FUNCTION_BLOCK FB_Cell
VAR_INPUT
END_VAR
VAR_OUTPUT
END_VAR
VAR
	eAutoMan					: E_AutoMan := E_AutoMan.AUTO;
	State						: E_CellState;
	
	// IO
	bStartBtn					AT %I* : BOOL;
	bStopBtn					AT %I* : BOOL;
	bPartPresentAtInfeed		AT %I* : BOOL;
	bPartPresentAtOutfeed		AT %I* : BOOL;
	
	{attribute 'TcAnalytics'}
	fFillRate					AT %Q* : LREAL := 2.5;
	
	// devices
	fbInfeedActuator			: FB_Actuator;
	fbOutfeedActuator			: FB_Actuator;
	fbInfeedConveyor			: FB_Axis;
	fbIndexConveyor				: FB_Axis;
	fbOutfeedConveyor			: FB_Axis;
	
	InfeedConveyor				: IAxis := fbInfeedConveyor;
	IndexConveyor				: IAxis := fbIndexConveyor;
	InfeedActuator				: IActuator := fbInfeedActuator;
	OutfeedActuator				: IActuator := fbOutfeedActuator;
	OutfeedConveyor				: IAxis := fbOutfeedConveyor;
	
	// stations
	fbBarcoder					: FB_BarcodeScanner;
	fbFiller					: FB_Filler;
	fbCapper					: FB_Capper;
	fbCheckWeigher				: FB_CheckWeigher;
	Stations					: ARRAY[0..3] OF IStation := [fbBarcoder, fbFiller, fbCapper, fbCheckWeigher];
	iStationCount				: DINT := 4;
	i							: DINT;
	
	bAllStationsReady			: BOOL;
	bCellPartPresent			: BOOL;
	bStationFaulted				: BOOL;
	tmrStationWait				: TON;
	bInFeeding					: BOOL;
	bIndexing					: BOOL;
	bOutfeeding					: BOOL;
	
	PartStatus					: ARRAY[0..3] OF ST_PartStatus;
	NewPart						: ST_PartStatus;
	
	{attribute 'TcAnalytics'}
	OutfeedPart					: ST_PartStatus;
	
	fIndexPosition				: LREAL;
	INDEX_DIST					: LREAL := 300.0;
	INDEX_VEL					: LREAL := 100.0;
	INFEED_VEL					: LREAL := 100.0;
	
	bStartReq					: BOOL;
	bStopReq					: BOOL;
	bInit 						: BOOL := TRUE;
	
	bFillRateTest				: BOOL;
	tmrFillRate					: TON;
END_VAR

METHOD PUBLIC CheckPart : BOOL
VAR_INPUT
	Status			: ST_PartStatus;
END_VAR
CheckPart := Status.bBarcodeStatus AND Status.bFillerStatus AND Status.bCapperStatus AND Status.bWeightStatus;
END_METHOD

METHOD PUBLIC Execute : PVOID
StationMgr();

IF eAutoMan = E_AutoMan.AUTO THEN
	
	CASE State OF
		
		E_CellState.STOPPED:
			
			IF bStartReq THEN
				State := E_CellState.IDLE_WAIT;
				bStartReq := FALSE;
			END_IF
			
		E_CellState.IDLE_WAIT:
		
			IF bPartPresentAtInfeed AND Stations[0] <> 0 
			AND (Stations[0].Ready AND NOT Stations[0].PartPresent) THEN
				State := E_CellState.FEED;
			END_IF
			
			IF bAllStationsReady AND bCellPartPresent THEN
				tmrStationWait(IN:=TRUE, PT:=T#500MS);
				IF tmrStationWait.Q THEN
					tmrStationWait(IN:=FALSE);
					State := E_CellState.INDEX;
				END_IF
			END_IF
			
			IF bStopReq THEN
				State := E_CellState.STOPPED;
				bStopReq := FALSE;
			END_IF
			
		E_CellState.FEED:
		
			IF NOT bInFeeding THEN
				MEMCPY(ADR(PartStatus[0]), ADR(NewPart), SIZEOF(ST_PartStatus));
				bInFeeding := TRUE;
			END_IF
			
			IF InfeedActuator.Cycle() THEN
				State := E_CellState.IDLE_WAIT;
				bInFeeding := FALSE;
			END_IF
			
		E_CellState.INDEX:
			
			IF NOT bIndexing THEN
				fIndexPosition := IndexConveyor.ActPosition + INDEX_DIST;
				bIndexing := TRUE;
			END_IF
			
			IF (IndexConveyor.MoveAbsolute(fIndexPosition, INDEX_VEL)) AND bIndexing THEN
				bIndexing := FALSE;
				OutfeedPart := PartStatus[3];
				MEMCPY(ADR(PartStatus[1]), ADR(PartStatus[0]), SIZEOF(ST_PartStatus)*3);
				MEMSET(ADR(PartStatus[0]), 0, SIZEOF(ST_PartStatus));
				State := E_CellState.IDLE_WAIT;
			END_IF
			
	END_CASE
	
	IF State <> E_CellState.STOPPED THEN
		
		InfeedConveyor.JogFwd(INFEED_VEL);
		OutfeedConveyor.JogFwd(INFEED_VEL);
		
		IF bPartPresentAtOutfeed THEN
			// bad part
			IF NOT CheckPart(OutfeedPart) THEN
				bOutFeeding := TRUE;
			END_IF
		END_IF
		IF bOutfeeding THEN
			IF OutfeedActuator.Cycle() THEN
				bOutfeeding := FALSE;
			END_IF
		END_IF
		
		IF bFillRateTest THEN
			tmrFillRate(IN:=NOT tmrFillRate.Q, PT:=T#20M); 
			IF tmrFillRate.Q THEN
				fFillRate := fFillRate + 0.05;
			END_IF
		END_IF
		
	ELSE
		InfeedConveyor.StopMove();
		OutfeedConveyor.StopMove();
	END_IF
	
END_IF

IF bStartBtn THEN
	bStopReq := FALSE;
	bStartReq := TRUE;
END_IF

IF bStopBtn THEN
	bStartReq := FALSE;
	bStopReq := TRUE;
END_IF
END_METHOD

METHOD PRIVATE StationMgr : PVOID
VAR_INPUT
END_VAR
IF iStationCount < 1 THEN
	RETURN;
END_IF

IF bInit THEN
	FOR i:= 0 TO iStationCount - 1 DO
		Stations[i].PartStatus := ADR(PartStatus[i]);
	END_FOR
	bInit := FALSE;
	bStartReq := TRUE;
END_IF

bAllStationsReady := TRUE;
bStationFaulted := FALSE;
bCellPartPresent := FALSE;

FOR i := 0 TO iStationCount - 1	DO
	IF (Stations[i] = 0) THEN
		CONTINUE;
	END_IF
	
	Stations[i].Execute();
	
	IF NOT Stations[i].Ready THEN
		bAllStationsReady := FALSE;
	END_IF
	
	IF Stations[i].Faulted THEN
		bStationFaulted := TRUE;
	END_IF
	
	IF Stations[i].PartPresent THEN
		bCellPartPresent := TRUE;
	END_IF
	
END_FOR
END_METHOD

END_FUNCTION_BLOCK

(* stored: Version 1.1.0.1, ProductVersion 3.1.4024.12
   POU FB_Cell: Id {94f7f691-4eab-4c8c-b55b-20327a9666cd}, SpecialFunc None
   Method CheckPart: Id {40737b5d-e3a6-42c5-9b7b-02e8083b82b0}
   Method Execute: Id {d7efdd70-bdc8-43b5-82c2-5ff6cb9ffaaa}
   Method StationMgr: Id {406f1cac-08f7-4834-90e0-c1f532d28c4c} *)
